// TIA Portal V19 export
FUNCTION "EDI" : Void   // FC12, LAD
{ S7_Optimized_Access := 'TRUE' }
// stored: SetENOAutomatically false
   VAR_TEMP   // added for the SCL form of the ladder/FBD networks
      _w1 : Bool;
   END_VAR
BEGIN

REGION Network 1: FEED PUMP
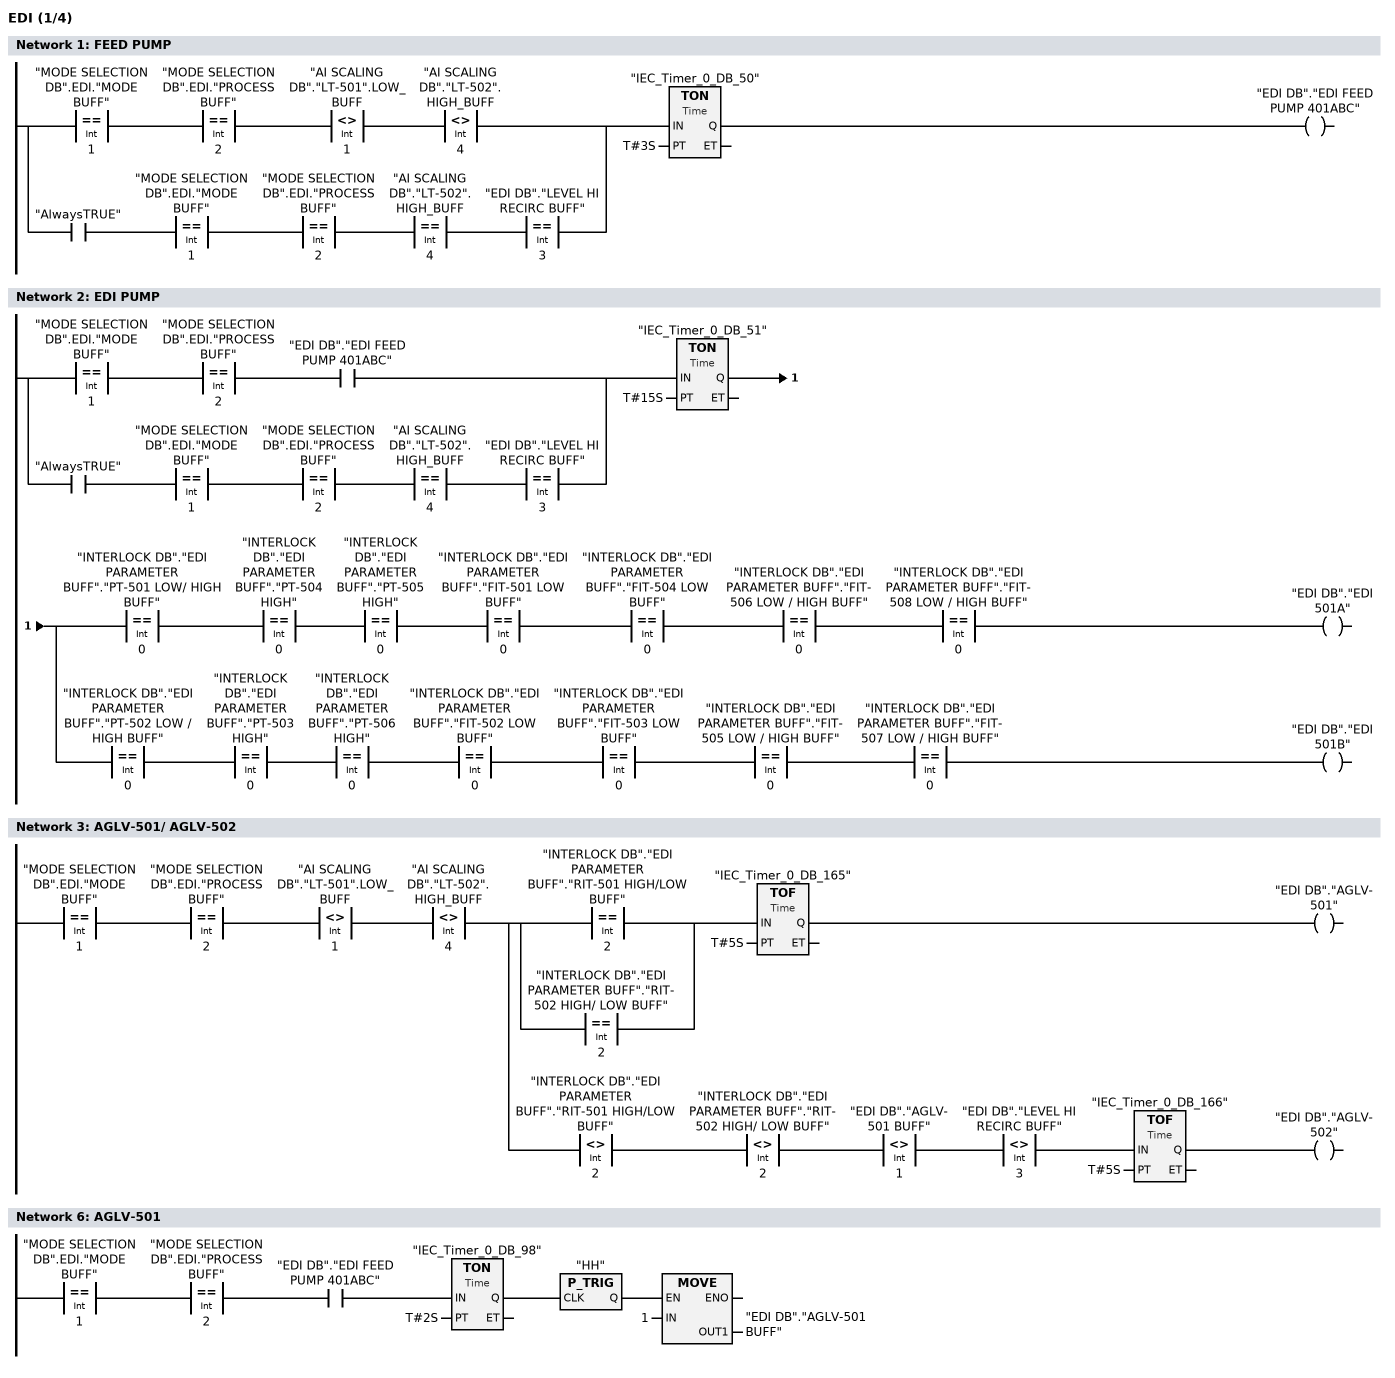
   RUNG wire#powerrail
      { S7_Templates := "SrcType := Int" } EQ_Contact(in1 := "MODE SELECTION DB".EDI."MODE BUFF", in2 := 1)
      { S7_Templates := "SrcType := Int" } EQ_Contact(in1 := "MODE SELECTION DB".EDI."PROCESS BUFF", in2 := 2)
      { S7_Templates := "SrcType := Int" } NE_Contact(in1 := "AI SCALING DB"."LT-501".LOW_BUFF, in2 := 1)
      { S7_Templates := "SrcType := Int" } NE_Contact(in1 := "AI SCALING DB"."LT-502".HIGH_BUFF, in2 := 4)
      wire#w1
      { S7_Templates := "time_type := Time" } "IEC_Timer_0_DB_50".TON(pt := T#3S, et =>)
      Coil( "EDI DB"."EDI FEED PUMP 401ABC" )
   END_RUNG
   RUNG wire#powerrail
      Contact( "AlwaysTRUE" )
      { S7_Templates := "SrcType := Int" } EQ_Contact(in1 := "MODE SELECTION DB".EDI."MODE BUFF", in2 := 1)
      { S7_Templates := "SrcType := Int" } EQ_Contact(in1 := "MODE SELECTION DB".EDI."PROCESS BUFF", in2 := 2)
      { S7_Templates := "SrcType := Int" } EQ_Contact(in1 := "AI SCALING DB"."LT-502".HIGH_BUFF, in2 := 4)
      { S7_Templates := "SrcType := Int" } EQ_Contact(in1 := "EDI DB"."LEVEL HI RECIRC BUFF", in2 := 3)
   END_RUNG wire#w1
   // the same network as SCL:
   "IEC_Timer_0_DB_50".TON(IN := (("MODE SELECTION DB".EDI."MODE BUFF" = 1) AND ("MODE SELECTION DB".EDI."PROCESS BUFF" = 2) AND ("AI SCALING DB"."LT-501".LOW_BUFF <> 1) AND ("AI SCALING DB"."LT-502".HIGH_BUFF <> 4)) OR ("AlwaysTRUE" AND ("MODE SELECTION DB".EDI."MODE BUFF" = 1) AND ("MODE SELECTION DB".EDI."PROCESS BUFF" = 2) AND ("AI SCALING DB"."LT-502".HIGH_BUFF = 4) AND ("EDI DB"."LEVEL HI RECIRC BUFF" = 3)),
                           PT := T#3S);
   "EDI DB"."EDI FEED PUMP 401ABC" := "IEC_Timer_0_DB_50".Q;
END_REGION

REGION Network 2: EDI PUMP
   RUNG wire#powerrail
      { S7_Templates := "SrcType := Int" } EQ_Contact(in1 := "MODE SELECTION DB".EDI."MODE BUFF", in2 := 1)
      { S7_Templates := "SrcType := Int" } EQ_Contact(in1 := "MODE SELECTION DB".EDI."PROCESS BUFF", in2 := 2)
      Contact( "EDI DB"."EDI FEED PUMP 401ABC" )
      wire#w1
      { S7_Templates := "time_type := Time" } "IEC_Timer_0_DB_51".TON(pt := T#15S, et =>)
      wire#w2
      { S7_Templates := "SrcType := Int" } EQ_Contact(in1 := "INTERLOCK DB"."EDI PARAMETER BUFF"."PT-501 LOW/ HIGH BUFF", in2 := 0)
      { S7_Templates := "SrcType := Int" } EQ_Contact(in1 := "INTERLOCK DB"."EDI PARAMETER BUFF"."PT-504 HIGH", in2 := 0)
      { S7_Templates := "SrcType := Int" } EQ_Contact(in1 := "INTERLOCK DB"."EDI PARAMETER BUFF"."PT-505 HIGH", in2 := 0)
      { S7_Templates := "SrcType := Int" } EQ_Contact(in1 := "INTERLOCK DB"."EDI PARAMETER BUFF"."FIT-501 LOW BUFF", in2 := 0)
      { S7_Templates := "SrcType := Int" } EQ_Contact(in1 := "INTERLOCK DB"."EDI PARAMETER BUFF"."FIT-504 LOW BUFF", in2 := 0)
      { S7_Templates := "SrcType := Int" } EQ_Contact(in1 := "INTERLOCK DB"."EDI PARAMETER BUFF"."FIT-506 LOW / HIGH BUFF", in2 := 0)
      { S7_Templates := "SrcType := Int" } EQ_Contact(in1 := "INTERLOCK DB"."EDI PARAMETER BUFF"."FIT-508 LOW / HIGH BUFF", in2 := 0)
      Coil( "EDI DB"."EDI 501A" )
   END_RUNG
   RUNG wire#powerrail
      Contact( "AlwaysTRUE" )
      { S7_Templates := "SrcType := Int" } EQ_Contact(in1 := "MODE SELECTION DB".EDI."MODE BUFF", in2 := 1)
      { S7_Templates := "SrcType := Int" } EQ_Contact(in1 := "MODE SELECTION DB".EDI."PROCESS BUFF", in2 := 2)
      { S7_Templates := "SrcType := Int" } EQ_Contact(in1 := "AI SCALING DB"."LT-502".HIGH_BUFF, in2 := 4)
      { S7_Templates := "SrcType := Int" } EQ_Contact(in1 := "EDI DB"."LEVEL HI RECIRC BUFF", in2 := 3)
   END_RUNG wire#w1
   RUNG wire#w2
      { S7_Templates := "SrcType := Int" } EQ_Contact(in1 := "INTERLOCK DB"."EDI PARAMETER BUFF"."PT-502 LOW / HIGH BUFF", in2 := 0)
      { S7_Templates := "SrcType := Int" } EQ_Contact(in1 := "INTERLOCK DB"."EDI PARAMETER BUFF"."PT-503 HIGH", in2 := 0)
      { S7_Templates := "SrcType := Int" } EQ_Contact(in1 := "INTERLOCK DB"."EDI PARAMETER BUFF"."PT-506 HIGH", in2 := 0)
      { S7_Templates := "SrcType := Int" } EQ_Contact(in1 := "INTERLOCK DB"."EDI PARAMETER BUFF"."FIT-502 LOW  BUFF", in2 := 0)
      { S7_Templates := "SrcType := Int" } EQ_Contact(in1 := "INTERLOCK DB"."EDI PARAMETER BUFF"."FIT-503 LOW BUFF", in2 := 0)
      { S7_Templates := "SrcType := Int" } EQ_Contact(in1 := "INTERLOCK DB"."EDI PARAMETER BUFF"."FIT-505 LOW / HIGH BUFF", in2 := 0)
      { S7_Templates := "SrcType := Int" } EQ_Contact(in1 := "INTERLOCK DB"."EDI PARAMETER BUFF"."FIT-507 LOW / HIGH BUFF", in2 := 0)
      Coil( "EDI DB"."EDI 501B" )
   END_RUNG
   // the same network as SCL:
   "IEC_Timer_0_DB_51".TON(IN := (("MODE SELECTION DB".EDI."MODE BUFF" = 1) AND ("MODE SELECTION DB".EDI."PROCESS BUFF" = 2) AND "EDI DB"."EDI FEED PUMP 401ABC") OR ("AlwaysTRUE" AND ("MODE SELECTION DB".EDI."MODE BUFF" = 1) AND ("MODE SELECTION DB".EDI."PROCESS BUFF" = 2) AND ("AI SCALING DB"."LT-502".HIGH_BUFF = 4) AND ("EDI DB"."LEVEL HI RECIRC BUFF" = 3)),
                           PT := T#15S);
   "EDI DB"."EDI 501A" := "IEC_Timer_0_DB_51".Q AND ("INTERLOCK DB"."EDI PARAMETER BUFF"."PT-501 LOW/ HIGH BUFF" = 0) AND ("INTERLOCK DB"."EDI PARAMETER BUFF"."PT-504 HIGH" = 0) AND ("INTERLOCK DB"."EDI PARAMETER BUFF"."PT-505 HIGH" = 0) AND ("INTERLOCK DB"."EDI PARAMETER BUFF"."FIT-501 LOW BUFF" = 0) AND ("INTERLOCK DB"."EDI PARAMETER BUFF"."FIT-504 LOW BUFF" = 0) AND ("INTERLOCK DB"."EDI PARAMETER BUFF"."FIT-506 LOW / HIGH BUFF" = 0) AND ("INTERLOCK DB"."EDI PARAMETER BUFF"."FIT-508 LOW / HIGH BUFF" = 0);
   "EDI DB"."EDI 501B" := "IEC_Timer_0_DB_51".Q AND ("INTERLOCK DB"."EDI PARAMETER BUFF"."PT-502 LOW / HIGH BUFF" = 0) AND ("INTERLOCK DB"."EDI PARAMETER BUFF"."PT-503 HIGH" = 0) AND ("INTERLOCK DB"."EDI PARAMETER BUFF"."PT-506 HIGH" = 0) AND ("INTERLOCK DB"."EDI PARAMETER BUFF"."FIT-502 LOW  BUFF" = 0) AND ("INTERLOCK DB"."EDI PARAMETER BUFF"."FIT-503 LOW BUFF" = 0) AND ("INTERLOCK DB"."EDI PARAMETER BUFF"."FIT-505 LOW / HIGH BUFF" = 0) AND ("INTERLOCK DB"."EDI PARAMETER BUFF"."FIT-507 LOW / HIGH BUFF" = 0);
END_REGION

REGION Network 3: AGLV-501/ AGLV-502
   RUNG wire#powerrail
      { S7_Templates := "SrcType := Int" } EQ_Contact(in1 := "MODE SELECTION DB".EDI."MODE BUFF", in2 := 1)
      { S7_Templates := "SrcType := Int" } EQ_Contact(in1 := "MODE SELECTION DB".EDI."PROCESS BUFF", in2 := 2)
      { S7_Templates := "SrcType := Int" } NE_Contact(in1 := "AI SCALING DB"."LT-501".LOW_BUFF, in2 := 1)
      { S7_Templates := "SrcType := Int" } NE_Contact(in1 := "AI SCALING DB"."LT-502".HIGH_BUFF, in2 := 4)
      wire#w1
      { S7_Templates := "SrcType := Int" } EQ_Contact(in1 := "INTERLOCK DB"."EDI PARAMETER BUFF"."RIT-501 HIGH/LOW BUFF", in2 := 2)
      wire#w2
      { S7_Templates := "time_type := Time" } "IEC_Timer_0_DB_165".TOF(pt := T#5S, et =>)
      Coil( "EDI DB"."AGLV-501" )
   END_RUNG
   RUNG wire#w1
      { S7_Templates := "SrcType := Int" } EQ_Contact(in1 := "INTERLOCK DB"."EDI PARAMETER BUFF"."RIT-502 HIGH/ LOW BUFF", in2 := 2)
   END_RUNG wire#w2
   RUNG wire#w1
      { S7_Templates := "SrcType := Int" } NE_Contact(in1 := "INTERLOCK DB"."EDI PARAMETER BUFF"."RIT-501 HIGH/LOW BUFF", in2 := 2)
      { S7_Templates := "SrcType := Int" } NE_Contact(in1 := "INTERLOCK DB"."EDI PARAMETER BUFF"."RIT-502 HIGH/ LOW BUFF", in2 := 2)
      { S7_Templates := "SrcType := Int" } NE_Contact(in1 := "EDI DB"."AGLV-501 BUFF", in2 := 1)
      { S7_Templates := "SrcType := Int" } NE_Contact(in1 := "EDI DB"."LEVEL HI RECIRC BUFF", in2 := 3)
      { S7_Templates := "time_type := Time" } "IEC_Timer_0_DB_166".TOF(pt := T#5S, et =>)
      Coil( "EDI DB"."AGLV-502" )
   END_RUNG
   // the same network as SCL:
   #_w1 := ("MODE SELECTION DB".EDI."MODE BUFF" = 1) AND ("MODE SELECTION DB".EDI."PROCESS BUFF" = 2) AND ("AI SCALING DB"."LT-501".LOW_BUFF <> 1) AND ("AI SCALING DB"."LT-502".HIGH_BUFF <> 4);
   "IEC_Timer_0_DB_165".TOF(IN := #_w1 AND (("INTERLOCK DB"."EDI PARAMETER BUFF"."RIT-501 HIGH/LOW BUFF" = 2) OR ("INTERLOCK DB"."EDI PARAMETER BUFF"."RIT-502 HIGH/ LOW BUFF" = 2)),
                           PT := T#5S);
   "EDI DB"."AGLV-501" := "IEC_Timer_0_DB_165".Q;
   "IEC_Timer_0_DB_166".TOF(IN := #_w1 AND ("INTERLOCK DB"."EDI PARAMETER BUFF"."RIT-501 HIGH/LOW BUFF" <> 2) AND ("INTERLOCK DB"."EDI PARAMETER BUFF"."RIT-502 HIGH/ LOW BUFF" <> 2) AND ("EDI DB"."AGLV-501 BUFF" <> 1) AND ("EDI DB"."LEVEL HI RECIRC BUFF" <> 3),
                           PT := T#5S);
   "EDI DB"."AGLV-502" := "IEC_Timer_0_DB_166".Q;
END_REGION

REGION Network 6: AGLV-501
   RUNG wire#powerrail
      { S7_Templates := "SrcType := Int" } EQ_Contact(in1 := "MODE SELECTION DB".EDI."MODE BUFF", in2 := 1)
      { S7_Templates := "SrcType := Int" } EQ_Contact(in1 := "MODE SELECTION DB".EDI."PROCESS BUFF", in2 := 2)
      Contact( "EDI DB"."EDI FEED PUMP 401ABC" )
      { S7_Templates := "time_type := Time" } "IEC_Timer_0_DB_98".TON(pt := T#2S, et =>)
      P_Trig( "HH" )
      Move(in := 1, out1 => "EDI DB"."AGLV-501 BUFF")
   END_RUNG
   // the same network as SCL:
   "IEC_Timer_0_DB_98".TON(IN := ("MODE SELECTION DB".EDI."MODE BUFF" = 1) AND ("MODE SELECTION DB".EDI."PROCESS BUFF" = 2) AND "EDI DB"."EDI FEED PUMP 401ABC",
                           PT := T#2S);
   #_w1 := "IEC_Timer_0_DB_98".Q AND NOT "HH";   // rising edge
   "HH" := "IEC_Timer_0_DB_98".Q;
   IF #_w1 THEN "EDI DB"."AGLV-501 BUFF" := 1; END_IF;
END_REGION

REGION Network 7
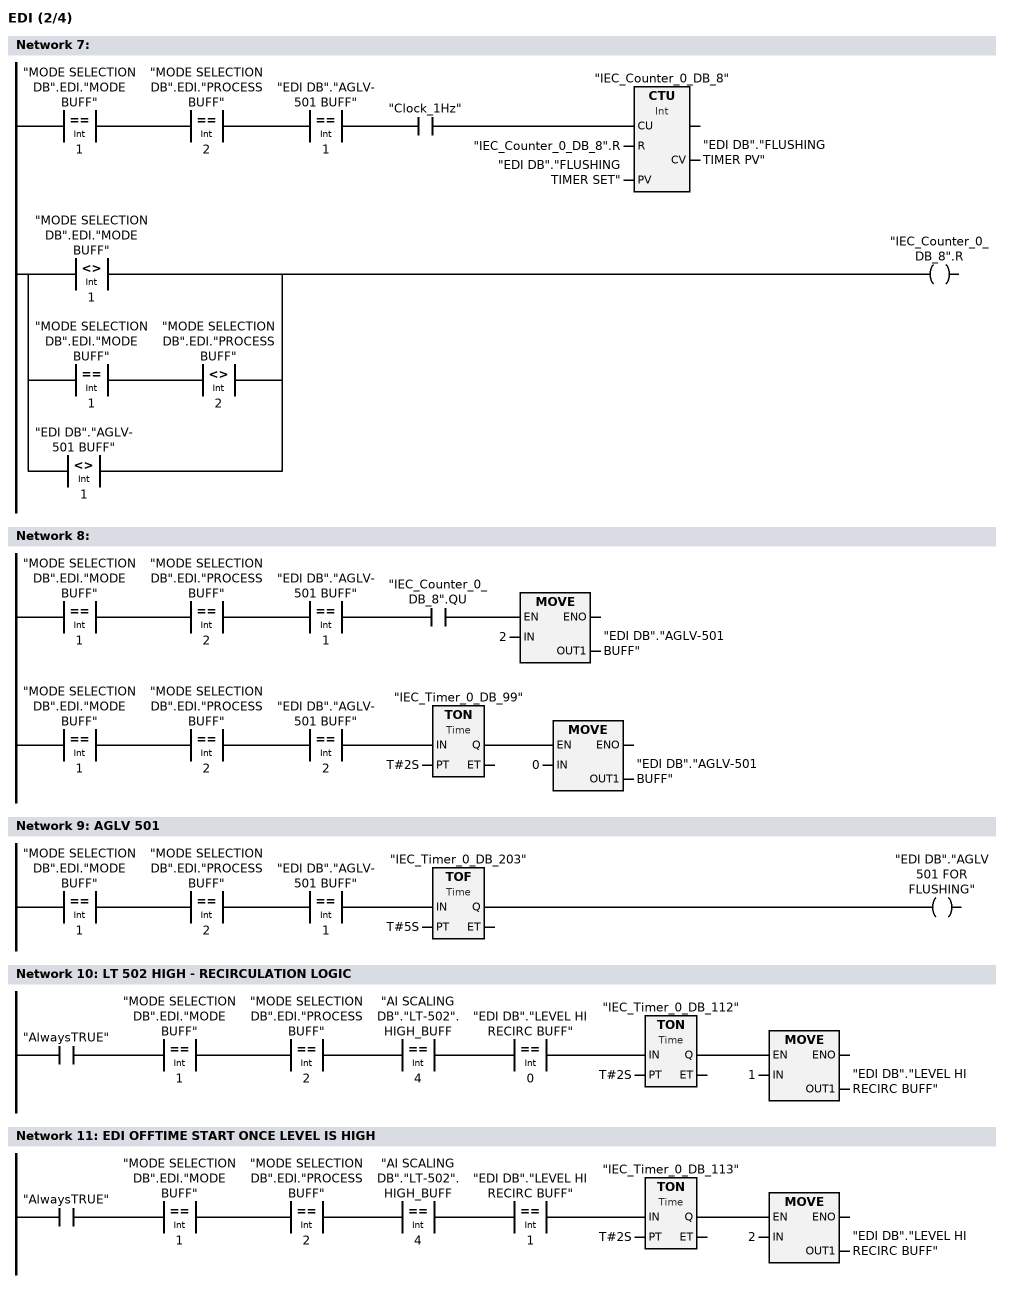
   RUNG wire#powerrail
      { S7_Templates := "SrcType := Int" } EQ_Contact(in1 := "MODE SELECTION DB".EDI."MODE BUFF", in2 := 1)
      { S7_Templates := "SrcType := Int" } EQ_Contact(in1 := "MODE SELECTION DB".EDI."PROCESS BUFF", in2 := 2)
      { S7_Templates := "SrcType := Int" } EQ_Contact(in1 := "EDI DB"."AGLV-501 BUFF", in2 := 1)
      Contact( "Clock_1Hz" )
      { S7_Templates := "value_type := Int" } "IEC_Counter_0_DB_8".CTU(r := "IEC_Counter_0_DB_8".R, pv := "EDI DB"."FLUSHING TIMER SET", cv => "EDI DB"."FLUSHING TIMER PV")
   END_RUNG
   RUNG wire#powerrail
      { S7_Templates := "SrcType := Int" } NE_Contact(in1 := "MODE SELECTION DB".EDI."MODE BUFF", in2 := 1)
      wire#w1
      Coil( "IEC_Counter_0_DB_8".R )
   END_RUNG
   RUNG wire#powerrail
      { S7_Templates := "SrcType := Int" } EQ_Contact(in1 := "MODE SELECTION DB".EDI."MODE BUFF", in2 := 1)
      { S7_Templates := "SrcType := Int" } NE_Contact(in1 := "MODE SELECTION DB".EDI."PROCESS BUFF", in2 := 2)
   END_RUNG wire#w1
   RUNG wire#powerrail
      { S7_Templates := "SrcType := Int" } NE_Contact(in1 := "EDI DB"."AGLV-501 BUFF", in2 := 1)
   END_RUNG wire#w1
   // the same network as SCL:
   "IEC_Counter_0_DB_8".CTU(CU := ("MODE SELECTION DB".EDI."MODE BUFF" = 1) AND ("MODE SELECTION DB".EDI."PROCESS BUFF" = 2) AND ("EDI DB"."AGLV-501 BUFF" = 1) AND "Clock_1Hz",
                           R := "IEC_Counter_0_DB_8".R,
                           PV := "EDI DB"."FLUSHING TIMER SET",
                           CV => "EDI DB"."FLUSHING TIMER PV");
   "IEC_Counter_0_DB_8".R := ("MODE SELECTION DB".EDI."MODE BUFF" <> 1) OR (("MODE SELECTION DB".EDI."MODE BUFF" = 1) AND ("MODE SELECTION DB".EDI."PROCESS BUFF" <> 2)) OR ("EDI DB"."AGLV-501 BUFF" <> 1);
END_REGION

REGION Network 8
   RUNG wire#powerrail
      { S7_Templates := "SrcType := Int" } EQ_Contact(in1 := "MODE SELECTION DB".EDI."MODE BUFF", in2 := 1)
      { S7_Templates := "SrcType := Int" } EQ_Contact(in1 := "MODE SELECTION DB".EDI."PROCESS BUFF", in2 := 2)
      { S7_Templates := "SrcType := Int" } EQ_Contact(in1 := "EDI DB"."AGLV-501 BUFF", in2 := 1)
      Contact( "IEC_Counter_0_DB_8".QU )
      Move(in := 2, out1 => "EDI DB"."AGLV-501 BUFF")
   END_RUNG
   RUNG wire#powerrail
      { S7_Templates := "SrcType := Int" } EQ_Contact(in1 := "MODE SELECTION DB".EDI."MODE BUFF", in2 := 1)
      { S7_Templates := "SrcType := Int" } EQ_Contact(in1 := "MODE SELECTION DB".EDI."PROCESS BUFF", in2 := 2)
      { S7_Templates := "SrcType := Int" } EQ_Contact(in1 := "EDI DB"."AGLV-501 BUFF", in2 := 2)
      { S7_Templates := "time_type := Time" } "IEC_Timer_0_DB_99".TON(pt := T#2S, et =>)
      Move(in := 0, out1 => "EDI DB"."AGLV-501 BUFF")
   END_RUNG
   // the same network as SCL:
   IF ("MODE SELECTION DB".EDI."MODE BUFF" = 1) AND ("MODE SELECTION DB".EDI."PROCESS BUFF" = 2) AND ("EDI DB"."AGLV-501 BUFF" = 1) AND "IEC_Counter_0_DB_8".QU THEN
       "EDI DB"."AGLV-501 BUFF" := 2;
   END_IF;
   "IEC_Timer_0_DB_99".TON(IN := ("MODE SELECTION DB".EDI."MODE BUFF" = 1) AND ("MODE SELECTION DB".EDI."PROCESS BUFF" = 2) AND ("EDI DB"."AGLV-501 BUFF" = 2),
                           PT := T#2S);
   IF "IEC_Timer_0_DB_99".Q THEN "EDI DB"."AGLV-501 BUFF" := 0; END_IF;
END_REGION

REGION Network 9: AGLV 501
   RUNG wire#powerrail
      { S7_Templates := "SrcType := Int" } EQ_Contact(in1 := "MODE SELECTION DB".EDI."MODE BUFF", in2 := 1)
      { S7_Templates := "SrcType := Int" } EQ_Contact(in1 := "MODE SELECTION DB".EDI."PROCESS BUFF", in2 := 2)
      { S7_Templates := "SrcType := Int" } EQ_Contact(in1 := "EDI DB"."AGLV-501 BUFF", in2 := 1)
      { S7_Templates := "time_type := Time" } "IEC_Timer_0_DB_203".TOF(pt := T#5S, et =>)
      Coil( "EDI DB"."AGLV 501 FOR FLUSHING" )
   END_RUNG
   // the same network as SCL:
   "IEC_Timer_0_DB_203".TOF(IN := ("MODE SELECTION DB".EDI."MODE BUFF" = 1) AND ("MODE SELECTION DB".EDI."PROCESS BUFF" = 2) AND ("EDI DB"."AGLV-501 BUFF" = 1),
                           PT := T#5S);
   "EDI DB"."AGLV 501 FOR FLUSHING" := "IEC_Timer_0_DB_203".Q;
END_REGION

REGION Network 10: LT 502 HIGH - RECIRCULATION LOGIC
   RUNG wire#powerrail
      Contact( "AlwaysTRUE" )
      { S7_Templates := "SrcType := Int" } EQ_Contact(in1 := "MODE SELECTION DB".EDI."MODE BUFF", in2 := 1)
      { S7_Templates := "SrcType := Int" } EQ_Contact(in1 := "MODE SELECTION DB".EDI."PROCESS BUFF", in2 := 2)
      { S7_Templates := "SrcType := Int" } EQ_Contact(in1 := "AI SCALING DB"."LT-502".HIGH_BUFF, in2 := 4)
      { S7_Templates := "SrcType := Int" } EQ_Contact(in1 := "EDI DB"."LEVEL HI RECIRC BUFF", in2 := 0)
      { S7_Templates := "time_type := Time" } "IEC_Timer_0_DB_112".TON(pt := T#2S, et =>)
      Move(in := 1, out1 => "EDI DB"."LEVEL HI RECIRC BUFF")
   END_RUNG
   // the same network as SCL:
   "IEC_Timer_0_DB_112".TON(IN := "AlwaysTRUE" AND ("MODE SELECTION DB".EDI."MODE BUFF" = 1) AND ("MODE SELECTION DB".EDI."PROCESS BUFF" = 2) AND ("AI SCALING DB"."LT-502".HIGH_BUFF = 4) AND ("EDI DB"."LEVEL HI RECIRC BUFF" = 0),
                           PT := T#2S);
   IF "IEC_Timer_0_DB_112".Q THEN "EDI DB"."LEVEL HI RECIRC BUFF" := 1; END_IF;
END_REGION

REGION Network 11: EDI OFFTIME START ONCE LEVEL IS HIGH
   RUNG wire#powerrail
      Contact( "AlwaysTRUE" )
      { S7_Templates := "SrcType := Int" } EQ_Contact(in1 := "MODE SELECTION DB".EDI."MODE BUFF", in2 := 1)
      { S7_Templates := "SrcType := Int" } EQ_Contact(in1 := "MODE SELECTION DB".EDI."PROCESS BUFF", in2 := 2)
      { S7_Templates := "SrcType := Int" } EQ_Contact(in1 := "AI SCALING DB"."LT-502".HIGH_BUFF, in2 := 4)
      { S7_Templates := "SrcType := Int" } EQ_Contact(in1 := "EDI DB"."LEVEL HI RECIRC BUFF", in2 := 1)
      { S7_Templates := "time_type := Time" } "IEC_Timer_0_DB_113".TON(pt := T#2S, et =>)
      Move(in := 2, out1 => "EDI DB"."LEVEL HI RECIRC BUFF")
   END_RUNG
   // the same network as SCL:
   "IEC_Timer_0_DB_113".TON(IN := "AlwaysTRUE" AND ("MODE SELECTION DB".EDI."MODE BUFF" = 1) AND ("MODE SELECTION DB".EDI."PROCESS BUFF" = 2) AND ("AI SCALING DB"."LT-502".HIGH_BUFF = 4) AND ("EDI DB"."LEVEL HI RECIRC BUFF" = 1),
                           PT := T#2S);
   IF "IEC_Timer_0_DB_113".Q THEN "EDI DB"."LEVEL HI RECIRC BUFF" := 2; END_IF;
END_REGION

REGION Network 12: EDI OFF TIME START
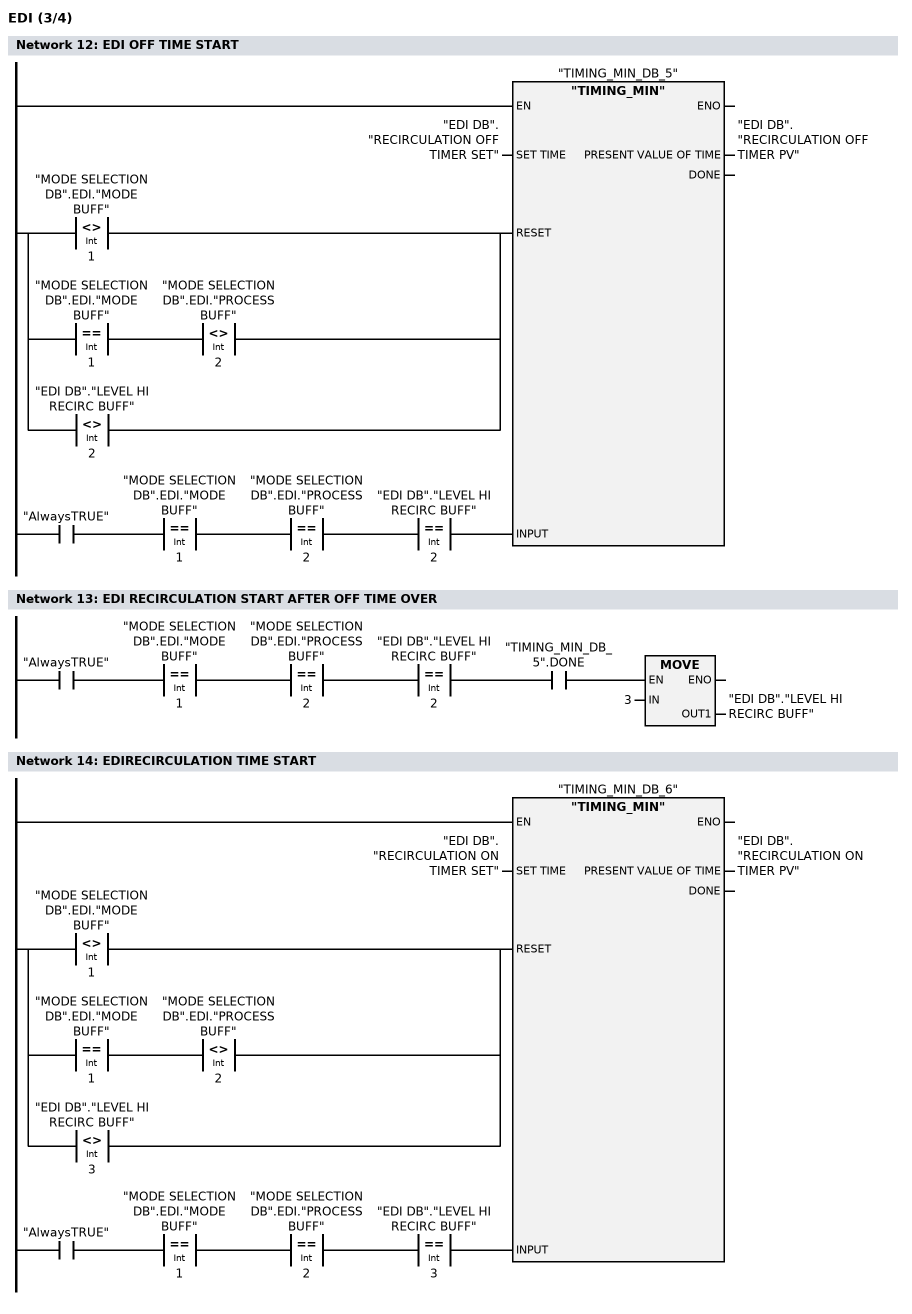
   RUNG wire#powerrail
      "TIMING_MIN_DB_5"(RESET := wire#w1, INPUT := wire#w2, "SET TIME" := "EDI DB"."RECIRCULATION OFF TIMER SET", "PRESENT VALUE OF TIME" => "EDI DB"."RECIRCULATION OFF TIMER PV", DONE =>)
   END_RUNG
   RUNG wire#powerrail
      { S7_Templates := "SrcType := Int" } NE_Contact(in1 := "MODE SELECTION DB".EDI."MODE BUFF", in2 := 1)
   END_RUNG wire#w1
   RUNG wire#powerrail
      { S7_Templates := "SrcType := Int" } EQ_Contact(in1 := "MODE SELECTION DB".EDI."MODE BUFF", in2 := 1)
      { S7_Templates := "SrcType := Int" } NE_Contact(in1 := "MODE SELECTION DB".EDI."PROCESS BUFF", in2 := 2)
   END_RUNG wire#w1
   RUNG wire#powerrail
      { S7_Templates := "SrcType := Int" } NE_Contact(in1 := "EDI DB"."LEVEL HI RECIRC BUFF", in2 := 2)
   END_RUNG wire#w1
   RUNG wire#powerrail
      Contact( "AlwaysTRUE" )
      { S7_Templates := "SrcType := Int" } EQ_Contact(in1 := "MODE SELECTION DB".EDI."MODE BUFF", in2 := 1)
      { S7_Templates := "SrcType := Int" } EQ_Contact(in1 := "MODE SELECTION DB".EDI."PROCESS BUFF", in2 := 2)
      { S7_Templates := "SrcType := Int" } EQ_Contact(in1 := "EDI DB"."LEVEL HI RECIRC BUFF", in2 := 2)
   END_RUNG wire#w2
   // the same network as SCL:
   "TIMING_MIN_DB_5"("SET TIME" := "EDI DB"."RECIRCULATION OFF TIMER SET",   // "TIMING_MIN"
                     RESET := ("MODE SELECTION DB".EDI."MODE BUFF" <> 1) OR (("MODE SELECTION DB".EDI."MODE BUFF" = 1) AND ("MODE SELECTION DB".EDI."PROCESS BUFF" <> 2)) OR ("EDI DB"."LEVEL HI RECIRC BUFF" <> 2),
                     INPUT := "AlwaysTRUE" AND ("MODE SELECTION DB".EDI."MODE BUFF" = 1) AND ("MODE SELECTION DB".EDI."PROCESS BUFF" = 2) AND ("EDI DB"."LEVEL HI RECIRC BUFF" = 2),
                     "PRESENT VALUE OF TIME" => "EDI DB"."RECIRCULATION OFF TIMER PV");
END_REGION

REGION Network 13: EDI RECIRCULATION START AFTER OFF TIME OVER
   RUNG wire#powerrail
      Contact( "AlwaysTRUE" )
      { S7_Templates := "SrcType := Int" } EQ_Contact(in1 := "MODE SELECTION DB".EDI."MODE BUFF", in2 := 1)
      { S7_Templates := "SrcType := Int" } EQ_Contact(in1 := "MODE SELECTION DB".EDI."PROCESS BUFF", in2 := 2)
      { S7_Templates := "SrcType := Int" } EQ_Contact(in1 := "EDI DB"."LEVEL HI RECIRC BUFF", in2 := 2)
      Contact( "TIMING_MIN_DB_5".DONE )
      Move(in := 3, out1 => "EDI DB"."LEVEL HI RECIRC BUFF")
   END_RUNG
   // the same network as SCL:
   IF "AlwaysTRUE" AND ("MODE SELECTION DB".EDI."MODE BUFF" = 1) AND ("MODE SELECTION DB".EDI."PROCESS BUFF" = 2) AND ("EDI DB"."LEVEL HI RECIRC BUFF" = 2) AND "TIMING_MIN_DB_5".DONE THEN
       "EDI DB"."LEVEL HI RECIRC BUFF" := 3;
   END_IF;
END_REGION

REGION Network 14: EDIRECIRCULATION TIME START
   RUNG wire#powerrail
      "TIMING_MIN_DB_6"(RESET := wire#w1, INPUT := wire#w2, "SET TIME" := "EDI DB"."RECIRCULATION ON TIMER SET", "PRESENT VALUE OF TIME" => "EDI DB"."RECIRCULATION ON TIMER PV", DONE =>)
   END_RUNG
   RUNG wire#powerrail
      { S7_Templates := "SrcType := Int" } NE_Contact(in1 := "MODE SELECTION DB".EDI."MODE BUFF", in2 := 1)
   END_RUNG wire#w1
   RUNG wire#powerrail
      { S7_Templates := "SrcType := Int" } EQ_Contact(in1 := "MODE SELECTION DB".EDI."MODE BUFF", in2 := 1)
      { S7_Templates := "SrcType := Int" } NE_Contact(in1 := "MODE SELECTION DB".EDI."PROCESS BUFF", in2 := 2)
   END_RUNG wire#w1
   RUNG wire#powerrail
      { S7_Templates := "SrcType := Int" } NE_Contact(in1 := "EDI DB"."LEVEL HI RECIRC BUFF", in2 := 3)
   END_RUNG wire#w1
   RUNG wire#powerrail
      Contact( "AlwaysTRUE" )
      { S7_Templates := "SrcType := Int" } EQ_Contact(in1 := "MODE SELECTION DB".EDI."MODE BUFF", in2 := 1)
      { S7_Templates := "SrcType := Int" } EQ_Contact(in1 := "MODE SELECTION DB".EDI."PROCESS BUFF", in2 := 2)
      { S7_Templates := "SrcType := Int" } EQ_Contact(in1 := "EDI DB"."LEVEL HI RECIRC BUFF", in2 := 3)
   END_RUNG wire#w2
   // the same network as SCL:
   "TIMING_MIN_DB_6"("SET TIME" := "EDI DB"."RECIRCULATION ON TIMER SET",   // "TIMING_MIN"
                     RESET := ("MODE SELECTION DB".EDI."MODE BUFF" <> 1) OR (("MODE SELECTION DB".EDI."MODE BUFF" = 1) AND ("MODE SELECTION DB".EDI."PROCESS BUFF" <> 2)) OR ("EDI DB"."LEVEL HI RECIRC BUFF" <> 3),
                     INPUT := "AlwaysTRUE" AND ("MODE SELECTION DB".EDI."MODE BUFF" = 1) AND ("MODE SELECTION DB".EDI."PROCESS BUFF" = 2) AND ("EDI DB"."LEVEL HI RECIRC BUFF" = 3),
                     "PRESENT VALUE OF TIME" => "EDI DB"."RECIRCULATION ON TIMER PV");
END_REGION

REGION Network 15: AGAIN OFF TIME START AFTER RECIRCULATION OVER
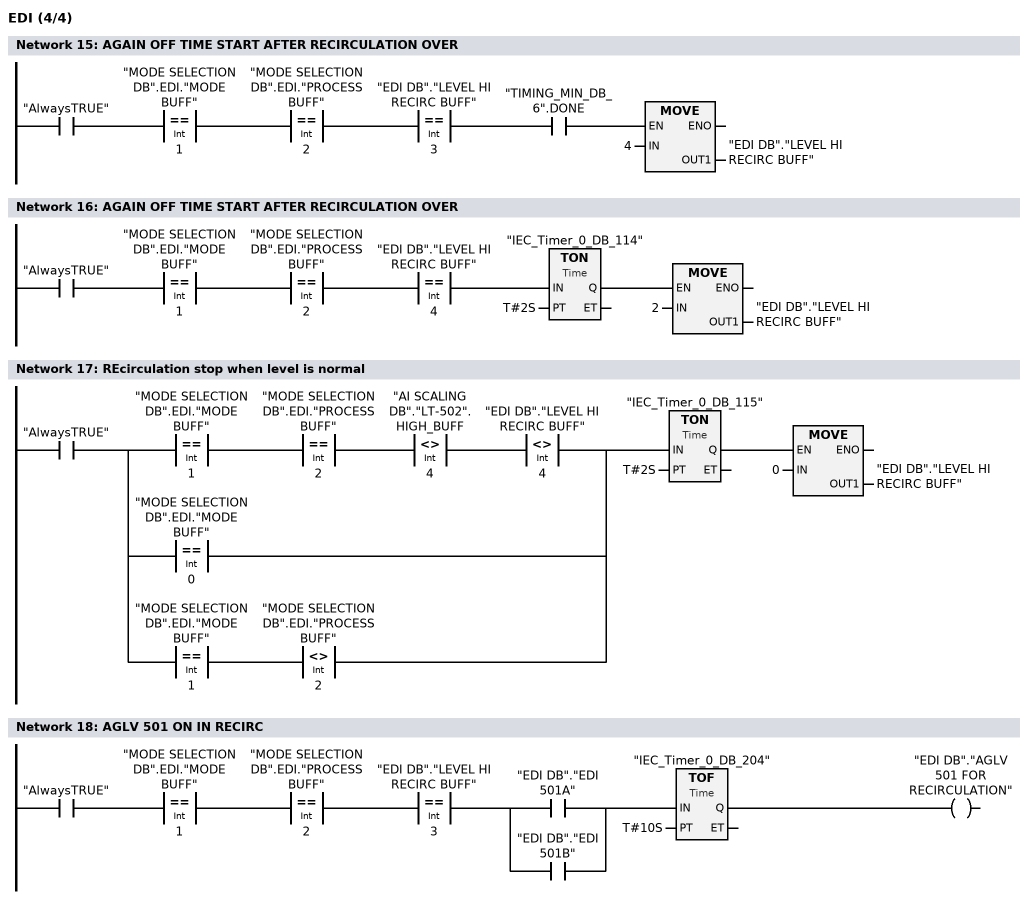
   RUNG wire#powerrail
      Contact( "AlwaysTRUE" )
      { S7_Templates := "SrcType := Int" } EQ_Contact(in1 := "MODE SELECTION DB".EDI."MODE BUFF", in2 := 1)
      { S7_Templates := "SrcType := Int" } EQ_Contact(in1 := "MODE SELECTION DB".EDI."PROCESS BUFF", in2 := 2)
      { S7_Templates := "SrcType := Int" } EQ_Contact(in1 := "EDI DB"."LEVEL HI RECIRC BUFF", in2 := 3)
      Contact( "TIMING_MIN_DB_6".DONE )
      Move(in := 4, out1 => "EDI DB"."LEVEL HI RECIRC BUFF")
   END_RUNG
   // the same network as SCL:
   IF "AlwaysTRUE" AND ("MODE SELECTION DB".EDI."MODE BUFF" = 1) AND ("MODE SELECTION DB".EDI."PROCESS BUFF" = 2) AND ("EDI DB"."LEVEL HI RECIRC BUFF" = 3) AND "TIMING_MIN_DB_6".DONE THEN
       "EDI DB"."LEVEL HI RECIRC BUFF" := 4;
   END_IF;
END_REGION

REGION Network 16: AGAIN OFF TIME START AFTER RECIRCULATION OVER
   RUNG wire#powerrail
      Contact( "AlwaysTRUE" )
      { S7_Templates := "SrcType := Int" } EQ_Contact(in1 := "MODE SELECTION DB".EDI."MODE BUFF", in2 := 1)
      { S7_Templates := "SrcType := Int" } EQ_Contact(in1 := "MODE SELECTION DB".EDI."PROCESS BUFF", in2 := 2)
      { S7_Templates := "SrcType := Int" } EQ_Contact(in1 := "EDI DB"."LEVEL HI RECIRC BUFF", in2 := 4)
      { S7_Templates := "time_type := Time" } "IEC_Timer_0_DB_114".TON(pt := T#2S, et =>)
      Move(in := 2, out1 => "EDI DB"."LEVEL HI RECIRC BUFF")
   END_RUNG
   // the same network as SCL:
   "IEC_Timer_0_DB_114".TON(IN := "AlwaysTRUE" AND ("MODE SELECTION DB".EDI."MODE BUFF" = 1) AND ("MODE SELECTION DB".EDI."PROCESS BUFF" = 2) AND ("EDI DB"."LEVEL HI RECIRC BUFF" = 4),
                           PT := T#2S);
   IF "IEC_Timer_0_DB_114".Q THEN "EDI DB"."LEVEL HI RECIRC BUFF" := 2; END_IF;
END_REGION

REGION Network 17: REcirculation stop when level is normal
   RUNG wire#powerrail
      Contact( "AlwaysTRUE" )
      wire#w1
      { S7_Templates := "SrcType := Int" } EQ_Contact(in1 := "MODE SELECTION DB".EDI."MODE BUFF", in2 := 1)
      { S7_Templates := "SrcType := Int" } EQ_Contact(in1 := "MODE SELECTION DB".EDI."PROCESS BUFF", in2 := 2)
      { S7_Templates := "SrcType := Int" } NE_Contact(in1 := "AI SCALING DB"."LT-502".HIGH_BUFF, in2 := 4)
      { S7_Templates := "SrcType := Int" } NE_Contact(in1 := "EDI DB"."LEVEL HI RECIRC BUFF", in2 := 4)
      wire#w2
      { S7_Templates := "time_type := Time" } "IEC_Timer_0_DB_115".TON(pt := T#2S, et =>)
      Move(in := 0, out1 => "EDI DB"."LEVEL HI RECIRC BUFF")
   END_RUNG
   RUNG wire#w1
      { S7_Templates := "SrcType := Int" } EQ_Contact(in1 := "MODE SELECTION DB".EDI."MODE BUFF", in2 := 0)
   END_RUNG wire#w2
   RUNG wire#w1
      { S7_Templates := "SrcType := Int" } EQ_Contact(in1 := "MODE SELECTION DB".EDI."MODE BUFF", in2 := 1)
      { S7_Templates := "SrcType := Int" } NE_Contact(in1 := "MODE SELECTION DB".EDI."PROCESS BUFF", in2 := 2)
   END_RUNG wire#w2
   // the same network as SCL:
   "IEC_Timer_0_DB_115".TON(IN := "AlwaysTRUE" AND ((("MODE SELECTION DB".EDI."MODE BUFF" = 1) AND ("MODE SELECTION DB".EDI."PROCESS BUFF" = 2) AND ("AI SCALING DB"."LT-502".HIGH_BUFF <> 4) AND ("EDI DB"."LEVEL HI RECIRC BUFF" <> 4)) OR ("MODE SELECTION DB".EDI."MODE BUFF" = 0) OR (("MODE SELECTION DB".EDI."MODE BUFF" = 1) AND ("MODE SELECTION DB".EDI."PROCESS BUFF" <> 2))),
                           PT := T#2S);
   IF "IEC_Timer_0_DB_115".Q THEN "EDI DB"."LEVEL HI RECIRC BUFF" := 0; END_IF;
END_REGION

REGION Network 18: AGLV 501 ON IN RECIRC
   RUNG wire#powerrail
      Contact( "AlwaysTRUE" )
      { S7_Templates := "SrcType := Int" } EQ_Contact(in1 := "MODE SELECTION DB".EDI."MODE BUFF", in2 := 1)
      { S7_Templates := "SrcType := Int" } EQ_Contact(in1 := "MODE SELECTION DB".EDI."PROCESS BUFF", in2 := 2)
      { S7_Templates := "SrcType := Int" } EQ_Contact(in1 := "EDI DB"."LEVEL HI RECIRC BUFF", in2 := 3)
      wire#w1
      Contact( "EDI DB"."EDI 501A" )
      wire#w2
      { S7_Templates := "time_type := Time" } "IEC_Timer_0_DB_204".TOF(pt := T#10S, et =>)
      Coil( "EDI DB"."AGLV 501 FOR RECIRCULATION" )
   END_RUNG
   RUNG wire#w1
      Contact( "EDI DB"."EDI 501B" )
   END_RUNG wire#w2
   // the same network as SCL:
   "IEC_Timer_0_DB_204".TOF(IN := "AlwaysTRUE" AND ("MODE SELECTION DB".EDI."MODE BUFF" = 1) AND ("MODE SELECTION DB".EDI."PROCESS BUFF" = 2) AND ("EDI DB"."LEVEL HI RECIRC BUFF" = 3) AND ("EDI DB"."EDI 501A" OR "EDI DB"."EDI 501B"),
                           PT := T#10S);
   "EDI DB"."AGLV 501 FOR RECIRCULATION" := "IEC_Timer_0_DB_204".Q;
END_REGION
END_FUNCTION
